// TIA Portal V21 export
// export: Created 2026-05-12T00:00:00.0000000Z, ExportSetting None
DATA_BLOCK "DB_HMI_Interface"   // DB200
{ S7_Optimized_Access := 'FALSE' }
   VAR
      CmdEnable : Bool := false;
      CmdDisable : Bool := false;
      CmdReset : Bool := false;
      CmdApply : Bool := false;
      _pad1_0_4 : Bool := false;
      _pad1_0_5 : Bool := false;
      _pad1_0_6 : Bool := false;
      _pad1_0_7 : Bool := false;
      StatusActive : Bool := false;
      StatusError : Bool := false;
      StatusWarning : Bool := false;
      StepNo : Int := 0;
      Setpoint : Real := 0.0;
      Actual : Real := 0.0;
      Output : Real := 0.0;
      OutputMin : Real := 0.0;
      OutputMax : Real := 100.0;
      CounterPreset : DInt := 10;
      CounterValue : DInt := 0;
   END_VAR
BEGIN
END_DATA_BLOCK
